INTERFACE I_MotionAxisNCDS402 EXTENDS I_MotionAxis, I_DS402Common

END_INTERFACE

(* stored: Version 1.1.0.1
   Itf I_MotionAxisNCDS402: Id {b75c273b-bf53-443f-ae0f-62773fbe19de} *)
